Staubli VAL3: TeachTool.pgx

public program TeachTool()
  local bool l_bBool
begin
  //示教工具
  //1.两点法进行示教
  //2.使用不拆工具法示教
  if TxtFile:bTeachToolMode
    CalTool:bUpLoad=false
    call CalTool:start()
     if CalTool:bUpLoad
      TxtFile:tCfg=CalTool:tTool
      call TxtFile:SaveCfg(l_bBool)
       if !l_bBool
        popUpMsg("保存失败")
      endIf
      call Kit:UpLoad()
    endIf

  else
    call  Teach2Tool()

  endIf

end
